// TIA Portal V20 export
TYPE "CC_Hmi_IO"
   STRUCT
      CC_RollsUp : Bool;
      CC_RollsDown : Bool;
      CC_ModulesUp : Bool;
      CC_ModulesDown : Bool;
      CC_Wibrating : Bool;
      CC_DriveRollerUp : Bool;
      CC_DriveRollerDown : Bool;
   END_STRUCT;
END_TYPE
